{attribute 'qualified_only'}
VAR_GLOBAL CONSTANT
	MAX_COLLEAGUES : INT := 6;
END_VAR

(* stored: Version 1.1.0.1, ProductVersion 3.1.4024.12
   GVL Param: Id {6782905d-b119-46bd-8557-d41cbec37753}, ParameterList True *)
